GLOBALCONSTANTS LED_COLOURS (* Global constants *)
  (* Standard: 61499-1; Description: Copyright (c) 2024 HR Agrartechnik GmbH This program and the accompanying materials are made available under the terms of the Eclipse Public License 2.0 which is available at https://www.eclipse.org/legal/epl-2.0/ SPDX-License-Identifier: EPL-2.0 *)
  (* Version 1.0, 2024-01-25, Franz Höpfinger, HR Agrartechnik GmbH *)
  PACKAGE logiBUS::io::DO_LED;
  VAR_GLOBAL CONSTANT
    LED_RED : UINT := 1;
    LED_YELLOW : UINT := 2;
    LED_ORANGE : UINT := 3;
    LED_GREEN : UINT := 4;
    LED_BLUE : UINT := 5;
    LED_WHITE : UINT := 6;
    LED_MAGENTA : UINT := 7;
    LED_CYAN : UINT := 8;
  END_VAR
END_GLOBALCONSTANTS
